// TIA Portal V19 export
TYPE "LEXCHANGETRAY_typeLogistics_deliver_interface"
// stored: Access Published
   STRUCT
      init : Bool;
      roller : "LEXCHANGETRAY_typeLogistics_toRollerDeliver";
   END_STRUCT;
END_TYPE
